# B&R Automation Studio project ControlPLC_DataDistribution (part 8)

#### VfLCRConnect.st - not currently in use
```iecst
FUNCTION_BLOCK VfLCRConnect

	IF (Execute) THEN

		// Trace the currently-active step; the most recent step is in array index [0].
		IF (Internal.Step <> Internal.StepTrace[0]) THEN
			FOR Internal.i := 99 TO 1 BY (-1) DO
				Internal.StepTrace[Internal.i] := Internal.StepTrace[Internal.i-1];
			END_FOR
			Internal.StepTrace[0] := Internal.Step;
		END_IF;

		// Main state machine
		CASE Internal.Step OF

			// Waiting for Execute
			vfLCR_CNCT_STEP_IDLE:
				Internal.Step := vfLCR_CNCT_STEP_CONNECT_LCR1;

			// Establish connection to local media where target file will be placed
			vfLCR_CNCT_STEP_CONNECT_LCR1:
				Internal.FB.DevLinkLocalLCR.pDevice := pLocalLCRDriveName;
				Internal.FB.DevLinkLocalLCR.pParam := pLocalLCRDrive;
				Internal.FB.DevLinkLocalLCR.enable := TRUE;
				Internal.Step := vfLCR_CNCT_STEP_CONNECT_LCR2;

			// Wait for successful connection
			vfLCR_CNCT_STEP_CONNECT_LCR2:
				IF (Internal.FB.DevLinkLocalLCR.status = ERR_OK) THEN
					Internal.FB.DevLinkLocalLCR.enable := FALSE;
					LocalLCRDriveHandle := Internal.FB.DevLinkLocalLCR.handle;
					Internal.Step := vfLCR_CNCT_STEP_DONE;

				ELSIF (Internal.FB.DevLinkLocalLCR.status <> ERR_FUB_BUSY) THEN
					Internal.FB.DevLinkLocalLCR.enable := FALSE;
					Internal.ErrorStep := Internal.Step;
					Error := TRUE;
					ErrorID := Internal.FB.DevLinkLocalLCR.status;
					Internal.Step := vfLCR_CNCT_STEP_DISCONNECT1;

				END_IF

				// Wait for incoming command
			vfLCR_CNCT_STEP_DONE:
				Done := TRUE;

				// Disconnect from all media
			vfLCR_CNCT_STEP_DISCONNECT1:
				IF (LocalLCRDriveHandle <> 0) THEN
					Internal.FB.DevUnlinkLocalLCR.handle := LocalLCRDriveHandle;
					Internal.FB.DevUnlinkLocalLCR.enable := TRUE;
				END_IF
				Internal.Step := vfLCR_CNCT_STEP_DISCONNECT2;

			vfLCR_CNCT_STEP_DISCONNECT2:
				// Wait for confirmation that both devices are unlinked
				IF ((Internal.FB.DevUnlinkLocalLCR.status = ERR_OK) OR (NOT Internal.FB.DevUnlinkLocalLCR.enable)) THEN
					LocalLCRDriveHandle := 0;
					Internal.Step := vfLCR_CNCT_STEP_ERROR;
				END_IF

			vfLCR_CNCT_STEP_ERROR:

				IF (ErrorReset) THEN
					Internal.Step := vfLCR_CNCT_STEP_ERROR_RESET;
				END_IF

			vfLCR_CNCT_STEP_ERROR_RESET:

		END_CASE

	ELSE // NOT Execute
		Internal.Step := vfLCR_CNCT_STEP_IDLE;
		Done := FALSE;
		Error := FALSE;
		ErrorID := ERR_OK;
		Internal.FB.DevLinkLocalLCR.enable := FALSE;
		Internal.FB.DevUnlinkLocalLCR.enable := FALSE;

	END_IF

	// Calling all FBs
	Internal.FB.DevLinkLocalLCR();
	Internal.FB.DevUnlinkLocalLCR();

END_FUNCTION_BLOCK
```

#### VfSMRFileSetup.st - not currently in use
```iecst
FUNCTION_BLOCK VfSMRFileSetup

	IF (Execute) THEN

		// Trace the currently-active step; the most recent step is in array index [0].
		IF (Internal.Step <> Internal.StepTrace[0]) THEN
			FOR Internal.index := 99 TO 1 BY (-1) DO
				Internal.StepTrace[Internal.index] := Internal.StepTrace[Internal.index-1];
			END_FOR
			Internal.StepTrace[0] := Internal.Step;
		END_IF;

		// Main state machine
		CASE Internal.Step OF

			// Waiting for execute command
			vfSMR_FILE_STEP_IDLE:
				Internal.Step := vfSMR_FILE_STEP_COPY_TO_SMR1;

					// Copy target file from remote media to local SMR CF card
			vfSMR_FILE_STEP_COPY_TO_SMR1:
				Internal.FB.FileCopy1.pSrcDev := pRemoteDriveName;
				Internal.FB.FileCopy1.pSrc := pPEFName;
				Internal.FB.FileCopy1.pDestDev := pLocalSMRDriveName;
				Internal.FB.FileCopy1.pDest := ADR('PEF.csv');
				Internal.FB.FileCopy1.option := fiOVERWRITE;
				Internal.FB.FileCopy1.enable := TRUE;
				Internal.Step := vfSMR_FILE_STEP_COPY_TO_SMR2;

				// Wait for completion of the copy operation
			vfSMR_FILE_STEP_COPY_TO_SMR2:
				IF (Internal.FB.FileCopy1.status = ERR_OK) THEN
					Internal.FB.FileCopy1.enable := FALSE;
					Internal.Step := vfSMR_FILE_STEP_COPY_TO_SMR3;

				ELSIF (Internal.FB.FileCopy1.status <> ERR_FUB_BUSY) THEN
					Internal.FB.FileCopy1.enable := FALSE;
					Internal.ErrorStep := Internal.Step;
					Error := TRUE;
					ErrorID := Internal.FB.FileCopy1.status;
					Internal.Step := vfSMR_FILE_STEP_ERROR;

				END_IF

			// Copy target file from remote media to local SMR CF card
			vfSMR_FILE_STEP_COPY_TO_SMR3:
				Internal.FB.FileCopy1.pSrcDev := pRemoteDriveName;
				Internal.FB.FileCopy1.pSrc := pFEFName;
				Internal.FB.FileCopy1.pDestDev := pLocalSMRDriveName;
				Internal.FB.FileCopy1.pDest := ADR('FEF.csv');
				Internal.FB.FileCopy1.option := fiOVERWRITE;
				Internal.FB.FileCopy1.enable := TRUE;
				Internal.Step := vfSMR_FILE_STEP_COPY_TO_SMR4;

			// Wait for completion of the copy operation
			vfSMR_FILE_STEP_COPY_TO_SMR4:
				IF (Internal.FB.FileCopy1.status = ERR_OK) THEN
					Internal.FB.FileCopy1.enable := FALSE;
					Internal.Step := vfSMR_FILE_STEP_COPY_TO_PTR1;

				ELSIF (Internal.FB.FileCopy1.status <> ERR_FUB_BUSY) THEN
					Internal.FB.FileCopy1.enable := FALSE;
					Internal.ErrorStep := Internal.Step;
					Error := TRUE;
					ErrorID := Internal.FB.FileCopy1.status;
					Internal.Step := vfSMR_FILE_STEP_ERROR;

				END_IF

				// Copy target file from local SMR CF card to local PTR CF card
			vfSMR_FILE_STEP_COPY_TO_PTR1:
				Internal.FB.FileCopy2.pSrcDev := pLocalSMRDriveName;
				Internal.FB.FileCopy2.pSrc := ADR('PEF.csv');
				Internal.FB.FileCopy2.pDestDev := pLocalPTRDriveName;
				Internal.FB.FileCopy2.pDest := ADR('PEF.csv');
				Internal.FB.FileCopy2.option := fiOVERWRITE;
				Internal.FB.FileCopy2.enable := TRUE;
				Internal.Step := vfSMR_FILE_STEP_COPY_TO_PTR2;

				// Wait for completion of the copy operation
			vfSMR_FILE_STEP_COPY_TO_PTR2:
				IF (Internal.FB.FileCopy2.status = ERR_OK) THEN
					Internal.FB.FileCopy2.enable := FALSE;
					Internal.Step := vfSMR_FILE_STEP_COPY_TO_LCR1;

				ELSIF (Internal.FB.FileCopy2.status <> ERR_FUB_BUSY) THEN
					Internal.FB.FileCopy2.enable := FALSE;
					Internal.ErrorStep := Internal.Step;
					Error := TRUE;
					ErrorID := Internal.FB.FileCopy2.status;
					Internal.Step := vfSMR_FILE_STEP_ERROR;

				END_IF

				// Copy target file from remote media to local LCR CF card
			vfSMR_FILE_STEP_COPY_TO_LCR1:
				Internal.FB.FileCopy3.pSrcDev := pLocalSMRDriveName;
				Internal.FB.FileCopy3.pSrc := ADR('FEF.csv');
				Internal.FB.FileCopy3.pDestDev := pLocalLCRDriveName;
				Internal.FB.FileCopy3.pDest := ADR('FEF.csv');
				Internal.FB.FileCopy3.option := fiOVERWRITE;
				Internal.FB.FileCopy3.enable := TRUE;
				Internal.Step := vfSMR_FILE_STEP_COPY_TO_LCR2;

				// Wait for completion of the copy operation
			vfSMR_FILE_STEP_COPY_TO_LCR2:
				IF (Internal.FB.FileCopy3.status = ERR_OK) THEN
					Internal.FB.FileCopy3.enable := FALSE;
					Internal.Step := vfSMR_FILE_STEP_DONE;

				ELSIF (Internal.FB.FileCopy3.status <> ERR_FUB_BUSY) THEN
					Internal.FB.FileCopy3.enable := FALSE;
					Internal.ErrorStep := Internal.Step;
					Error := TRUE;
					ErrorID := Internal.FB.FileCopy3.status;
					Internal.Step := vfSMR_FILE_STEP_ERROR;

				END_IF

				// We're officially done.
			vfSMR_FILE_STEP_DONE:
				Done := TRUE;

			vfSMR_FILE_STEP_ERROR:

				IF (ErrorReset) THEN
					Internal.Step := vfSMR_FILE_STEP_ERROR_RESET;
				END_IF

			vfSMR_FILE_STEP_ERROR_RESET:

		END_CASE

	ELSE // NOT Execute
		Internal.Step := vfSMR_FILE_STEP_IDLE;
		Done := FALSE;
		Error := FALSE;
		ErrorID := ERR_OK;
		Internal.FB.FileCopy1.enable := FALSE;
		Internal.FB.FileCopy2.enable := FALSE;
		Internal.FB.FileCopy3.enable := FALSE;
	END_IF

	// Calling all FBs
	Internal.FB.FileCopy1();
	Internal.FB.FileCopy2();
	Internal.FB.FileCopy3();
END_FUNCTION_BLOCK
```

#### HelperFunctions.st
```iecst
FUNCTION GetNextString

	// Return error if function is called with missing parameters.
	IF (pAdrData = 0) OR (pParameter = 0) THEN
		GetNextString := vfp_ERR_NULL_POINTER;
		RETURN;
	END_IF

	// AdrData is the starting address of the data to be parsed.
	AdrData ACCESS pAdrData;
	ParameterValue ACCESS pParameter;

	FOR index := 0 TO (vfp_MAX_CHARS_PER_STRING_VALUE - 1) DO

		// Examine one character at a time, beginning at the starting address.
		CharVal ACCESS (AdrData + index);

		// If a NULL character is encountered, return with an error code.
		IF (CharVal = 0) THEN
			AdrData := AdrData + index;
			GetNextString := vfp_ERR_MISSING_DATA;
			RETURN;

			// When a carriage return or delimiter character is found...
		ELSIF ((CharVal = vfp_CHAR_COMMA) OR (CharVal = vfp_CHAR_CARRIAGE_RETURN)) THEN

			// If no data is present, return an error code indicating missing data (before delimiter) or end of line.
			IF (index = 0) THEN
				IF (CharVal = vfp_CHAR_COMMA) THEN
					AdrData := AdrData + index + 1;
					GetNextString := vfp_ERR_MISSING_DATA;
				ELSE
					AdrData := AdrData + index;
					GetNextString := vfp_ERR_EOL_REACHED;
				END_IF
				RETURN;

				// Otherwise, return the string in ParameterValue.
			ELSE
				brsmemset(ADR(TempString), 0, SIZEOF(TempString));
				brsmemcpy(ADR(TempString), AdrData, index);
				ParameterValue := TempString;

				// If a carriage return was found, return the the address of the CURRENT character for further processing.
				IF (CharVal = vfp_CHAR_CARRIAGE_RETURN) THEN
					AdrData := AdrData + index;
					GetNextString := vfp_ERR_EOL_REACHED;
					// Otherwise, a delimiter was found, so return the address of the NEXT character for further processing.
				ELSE
					AdrData := AdrData + index + 1;
					GetNextString := vfp_ERR_OK;
				END_IF
				RETURN;

			END_IF

		END_IF

	END_FOR

	// No delimiters were found in the search range.
	AdrData := AdrData + index;
	GetNextString := vfp_ERR_NO_DELIMITER;

END_FUNCTION

FUNCTION GetNextParameter

	// Return error if function is called with missing parameters.
	IF (pAdrData = 0) OR (pParameter = 0) THEN
		GetNextParameter := vfp_ERR_NULL_POINTER;
		RETURN;
	END_IF

	// AdrData is the starting address of the data to be parsed.
	AdrData ACCESS pAdrData;
	ParameterValue ACCESS pParameter;

	FOR index := 0 TO (vfp_MAX_CHARS_PER_NUMERIC_VALUE - 1) DO

		// Examine one character at a time, beginning at the starting address.
		CharVal ACCESS (AdrData + index);

		// If a NULL character is encountered, return with an error code.
		IF (CharVal = 0) THEN
			AdrData := AdrData + index;
			GetNextParameter := vfp_ERR_MISSING_DATA;
			RETURN;

			// When a carriage return or delimiter character is found...
		ELSIF ((CharVal = vfp_CHAR_COMMA) OR (CharVal = vfp_CHAR_CARRIAGE_RETURN)) THEN

			// If no data is present, return an error code indicating missing data (before delimiter) or end of line.
			IF (index = 0) THEN
				IF (CharVal = vfp_CHAR_COMMA) THEN
					AdrData := AdrData + index + 1;
					GetNextParameter := vfp_ERR_MISSING_DATA;
				ELSE
					AdrData := AdrData + index;
					GetNextParameter := vfp_ERR_EOL_REACHED;
				END_IF
				RETURN;

				// Otherwise, convert the numeric string to a floating point value and return it in the ParameterValue.
			ELSE
				brsmemset(ADR(TempString), 0, SIZEOF(TempString));
				brsmemcpy(ADR(TempString), AdrData, index);
				ParameterValue := brsatod(ADR(TempString));

				// If a carriage return was found, return the the address of the CURRENT character for further processing.
				IF (CharVal = vfp_CHAR_CARRIAGE_RETURN) THEN
					AdrData := AdrData + index;
					GetNextParameter := vfp_ERR_EOL_REACHED;
					// Otherwise, a delimiter was found, so return the address of the NEXT character for further processing.
				ELSE
					AdrData := AdrData + index + 1;
					GetNextParameter := vfp_ERR_OK;
				END_IF
				RETURN;

			END_IF

			// If a non-numerical value was found...
			// HACK: Spaces are ignored here; this is just a hack
		ELSIF (((CharVal < vfp_CHAR_DIGIT_0) OR (CharVal > vfp_CHAR_DIGIT_9)) AND (CharVal <> vfp_CHAR_DECIMAL_POINT) AND (CharVal <> vfp_CHAR_SPACE)) THEN
			// Return the address of the CURRENT character for further processing.
			AdrData := AdrData + index;
			GetNextParameter := vfp_ERR_NON_NUMERICAL;
			RETURN;
		END_IF

	END_FOR

	// No delimiters were found in the search range.
	AdrData := AdrData + index;
	GetNextParameter := vfp_ERR_NO_DELIMITER;

END_FUNCTION

FUNCTION FindNextLineStart

	// Return error if function is called with missing parameters.
	IF (pAdrData = 0) THEN
		FindNextLineStart := vfp_ERR_NULL_POINTER;
		RETURN;
	END_IF
	IF (MaxBytes = 0) THEN
		FindNextLineStart := vfp_ERR_INVALID_PARAMETER;
		RETURN;
	END_IF

	// AdrData is the starting address of the data to be parsed.
	AdrData ACCESS pAdrData;
	index := 0;

	// Examine one character at a time, searching for a line feed character (or end of buffer).
	REPEAT
		CharVal ACCESS (AdrData + index);
		index := index + 1;
		UNTIL
		(CharVal = vfp_CHAR_LINE_FEED) OR (CharVal = 0) OR (index >= MaxBytes)
	END_REPEAT;

	// If a line feed is found, return the address of the NEXT character for further processing.
	IF (CharVal = vfp_CHAR_LINE_FEED) THEN
		AdrData := AdrData + index;
		FindNextLineStart := vfp_ERR_OK;
	ELSE
		AdrData := AdrData + index;
		FindNextLineStart := vfp_ERR_MISSING_DATA;
	END_IF

END_FUNCTION

FUNCTION FindNextTrajectoryStart

	// Return error if function is called with missing parameters.
	IF (pAdrData = 0) THEN
		FindNextTrajectoryStart := vfp_ERR_NULL_POINTER;
		RETURN;
	END_IF
	IF (MaxBytes = 0) THEN
		FindNextTrajectoryStart := vfp_ERR_INVALID_PARAMETER;
		RETURN;
	END_IF

	// AdrData is the starting address of the data to be parsed.
	AdrData ACCESS pAdrData;
	index := 0;

	// Examine one character at a time, searching for a line feed character (or end of buffer).
	REPEAT
		CharVal ACCESS (AdrData + index);
		index := index + 1;
		UNTIL
		(CharVal = vfp_CHAR_TRAJECTORY_HDR) OR (CharVal = 0) OR (index >= MaxBytes)
	END_REPEAT;

	// If a trajectory header is found, return the address of the CURRENT character for further processing.
	IF (CharVal = vfp_CHAR_TRAJECTORY_HDR) THEN
		AdrData := AdrData + index - 1;
		FindNextTrajectoryStart := vfp_ERR_OK;
	ELSE
		AdrData := AdrData + index - 1;
		FindNextTrajectoryStart := vfp_ERR_MISSING_DATA;
	END_IF

END_FUNCTION

FUNCTION GetSystemErrorText

	CASE (ErrorID) OF

		0, vfp_ERR_OK:
			ErrorText := 'No Error';
		vfp_ERR_EOL_REACHED:
			ErrorText := 'Unexpected end-of-line encountered';
		vfp_ERR_NO_MORE_LINES:
			ErrorText := 'No more lines in file';
		vfp_ERR_NULL_POINTER:
			ErrorText := 'Null pointer in function call';
		vfp_ERR_INVALID_PARAMETER:
			ErrorText := 'Invalid parameter in function call';
		vfp_ERR_NO_DELIMITER:
			ErrorText := 'Required delimiter missing';
		vfp_ERR_MISSING_DATA:
			ErrorText := 'Required data missing';
		vfp_ERR_NON_NUMERICAL:
			ErrorText := 'Non-numerical value detected';
		vfp_ERR_WRONG_NUM_STATES:
			ErrorText := 'Wrong number of laser states';
		vfp_ERR_BAD_HEADER:
			ErrorText := 'Bad file header';
		vfp_ERR_HEADER_INVALID_NUM_TRAJ:
			ErrorText := 'Invlaid number of trajectories';
		vfp_ERR_BUFFER_SIZE:
			ErrorText := 'Inadequate buffer size declaration';
		vfp_ERR_FATAL_SYSTEM_ERROR:
			ErrorText := 'Fatal system error (recovery not possible)';

		fiERR_FILE_NOT_FOUND:
			ErrorText := 'File does not exist';

		ELSE
			ErrorText := 'no error text available';
	END_CASE

	GetSystemErrorText := TRUE;

END_FUNCTION
```

- Visualisation Logical/mappView (not shown)

Listed in the project but not available here: Logical/MachineControl/PiperModuleTemplate, Logical/MachineControl/MachineMode/MachineMode.typ, Logical/MachineControl/MachineMode/MachineMode.var, Logical/Automation/SFCControl/PiperModule.var, Logical/Automation/DataDistributionSFC/Init.st, Logical/ProcessControl/VFLCR/VFPTR_System/Types.typ, Logical/ProcessControl/VFLCR/VFPTR_System/Variables.var, Logical/ProcessControl/VFLCR/VFPTR_System/PiperModule.var, Logical/ProcessControl/VFLCR/VFPTR_System/PiperInterface.st, Logical/DataManagement/RecipeManagement.var, Logical/DataManagement/PrintJobManagement/Opcua.typ, Logical/DataManagement/PrintJobManagement/Variables.var, Logical/DataManagement/PrintJobManagement/PrintJobManagement/Variables.var, Logical/DataManagement/PrintJobManagement/BuildDistributor/Types.typ, Logical/DataManagement/PrintJobManagement/BuildDistributor/Variables.var, Logical/DataManagement/PrintJobManagement/BuildDistributor/PiperModule.var, Logical/DataManagement/PrintJobManagement/BuildDistributor/Simulation.st, Logical/Infrastructure/FirstInitProg/FirstInitProg.typ, Logical/Libraries/VF/VF_COMMON/VF_COMMON.var, Logical/Libraries/VF/ToolBox/Types.typ, Logical/Libraries/VF/ToolBox/Constants.var, Logical/Libraries/VF/VFValve/Constants.var, Logical/Libraries/Testing
